// Mitsubishi GX Works2 project: LIGAR-DESLIGAR COM PULSE   PLC: Q03UDV

PROGRAM MAIN
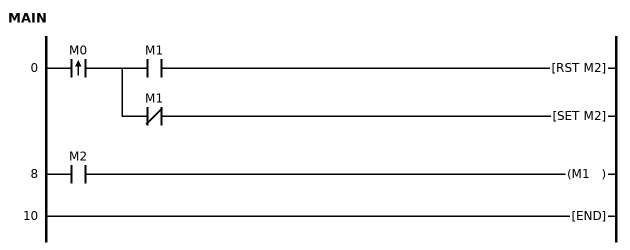
0     LDP     M0
      MPS
      AND     M1
      RST     M2
      MPP
      ANI     M1
      SET     M2
8     LD      M2
      OUT     M1
10    END
END_PROGRAM
